PROGRAM PRG_VALVES
VAR
    //Rough lines VRC external interlocks
    bROUGH1_VRC_01_ILK : BOOL;
    bROUGH2_VRC_01_ILK : BOOL;
    bROUGH2_VRC_02_ILK : BOOL;
    bROUGH1_VRC_01_Override : BOOL;
    bROUGH2_VRC_01_Override : BOOL;
    bROUGH2_VRC_02_Override : BOOL;
    bCAT1_VRC_01_ILK : BOOL;
    bDP1_VRC_01_ILK : BOOL;
    bDP1_VRC_02_ILK : BOOL;

    bCAT1_DisableDiffIlk : BOOL;

    //dummy FF output to use in VGC_2S function
    dummy_FFFO : FB_HardwareFFOutput;
    dummy_fbArbiter1 : FB_Arbiter(1);
END_VAR

(**Gas Injection Valves**)
DREAM_DP1_VRC_01(i_stUSG := DREAM_NC_GPI_01.PG,
                 i_stDSG := DREAM_DP1_GPI_01.PG,
                 i_xDis_DPIlk := FALSE,
                 i_xEPS_OK := TRUE,
                 i_xPMPS_OK := TRUE,
                 i_xReset := FALSE,
                 i_xExt_OK := TRUE,
                 i_xOverrideMode := bSystemOverrideMode,
                 io_fbFFHWO := dummy_FFFO,
                 fbArbiter := dummy_fbArbiter1,
                 i_sDevName := 'DREAM-DP1-VRC-01');

//DP1_VRC_02 Interlock evaluation NOTE: Normally OPEN Valve!!
bDP1_VRC_02_ILK := DREAM_DP1_VRC_01.iq_stValve.i_xOpnLS; //Interlock changed for this valve to only gets interlocked by DREAM_DP1_VRC_01 valve

DREAM_DP1_VRC_02(i_xExtILK_OK := bDP1_VRC_02_ILK, i_xOverrideMode := bSystemOverrideMode); //Normally open valve

(**Catcher valve**)
//Evaluate if Diff Interlock is disabled
bCAT1_DisableDiffIlk := NOT GVL_VAC_GAUGES.stDREAM_MC_GAUGE.xPRESS_OK OR NOT DREAM_CAT1_GHC_01.IG.xPRESS_OK;

//CAT1_VRC_01 Interlock evaluation
IF bCAT1_DisableDiffIlk THEN
    bCAT1_VRC_01_ILK := bMCPumpsRunning AND bCATPumpsRunning AND
                        ((GVL_VAC_GAUGES.stDREAM_MC_GAUGE.xPRESS_OK AND GVL_VAC_GAUGES.stDREAM_MC_GAUGE.rPRESS < 5e-4) OR (DREAM_MC_GPI_01.PG.xPRESS_OK AND DREAM_MC_GPI_01.PG.rPRESS < 5e-4)) AND
                        ((DREAM_CAT1_GHC_01.IG.xPRESS_OK AND DREAM_CAT1_GHC_01.IG.rPRESS < 5e-4) OR (DREAM_ROUGH2_GPI_03.PG.xPRESS_OK AND DREAM_ROUGH2_GPI_03.PG.rPRESS < 1e-3));
ELSE
    bCAT1_VRC_01_ILK := bCATPumpsRunning;
END_IF

//DREAM_CAT1_VRC_01(i_xExtILK_OK := bCAT1_VRC_01_ILK, i_xOverrideMode := bSystemOverrideMode);
DREAM_CAT1_VRC_01(i_stUSG := GVL_VAC_GAUGES.stDREAM_MC_GAUGE,
                  i_stDSG := DREAM_CAT1_GHC_01.IG,
                  i_xDis_DPIlk := bCAT1_DisableDiffIlk,
                  i_xEPS_OK := TRUE,
                  i_xPMPS_OK := TRUE,
                  i_xReset := FALSE,
                  i_xExt_OK := bCAT1_VRC_01_ILK,
                  i_xOverrideMode := bSystemOverrideMode,
                  io_fbFFHWO := dummy_FFFO,
                  fbArbiter := dummy_fbArbiter1,
                  i_sDevName := 'DREAM-CAT1-VRC-01');

(**Roughing Valves**)
//Interlock evaluation
bROUGH1_VRC_01_ILK := //DREAM_ROUGH1_GPI_01.PG.rPRESS < 5E-3 AND DREAM_ROUGH1_GPI_01.PG.xPRESS_OK AND
                      DREAM_ROUGH1_VFV_01.iq_stVFN.rReqPosition = 0.0 AND
                      DREAM_ROUGH1_VFV_02.iq_stVFN.rReqPosition = 0.0 AND
                      DREAM_ROUGH1_VRC_10.iq_stValve.i_xClsLS; //Interlocked with manifold roughing valve as well

bROUGH2_VRC_01_ILK := //DREAM_ROUGH2_GPI_01.PG.rPRESS < 5E-3 AND DREAM_ROUGH2_GPI_01.PG.xPRESS_OK AND
                      DREAM_ROUGH2_VFV_01.iq_stVFN.rReqPosition = 0.0 AND
                      DREAM_ROUGH2_VFV_02.iq_stVFN.rReqPosition = 0.0;

bROUGH2_VRC_02_ILK := //DREAM_ROUGH2_GPI_01.PG.rPRESS < 5E-3 AND DREAM_ROUGH2_GPI_01.PG.xPRESS_OK AND
                      DREAM_ROUGH2_VFV_01.iq_stVFN.rReqPosition = 0.0 AND
                      DREAM_ROUGH2_VFV_03.iq_stVFN.rReqPosition = 0.0;

bROUGH1_VRC_01_Override := bSystemOverrideMode AND
                           DREAM_ROUGH1_VFV_01.iq_stVFN.rReqPosition = 0.0 AND
                           DREAM_ROUGH1_VFV_02.iq_stVFN.rReqPosition = 0.0;

bROUGH2_VRC_01_Override := bSystemOverrideMode AND
                           DREAM_ROUGH2_VFV_01.iq_stVFN.rReqPosition = 0.0 AND
                           DREAM_ROUGH2_VFV_02.iq_stVFN.rReqPosition = 0.0;

bROUGH2_VRC_02_Override := bSystemOverrideMode AND
                           DREAM_ROUGH2_VFV_01.iq_stVFN.rReqPosition = 0.0 AND
                           DREAM_ROUGH2_VFV_03.iq_stVFN.rReqPosition = 0.0;

DREAM_ROUGH1_VRC_01(i_stUSG := DREAM_ROUGH1_GPI_01.PG,
                    i_stDSG := DREAM_ROUGH1_GPI_02.PG,
                    i_xDis_DPIlk := FALSE,
                    i_xEPS_OK := TRUE,
                    i_xPMPS_OK := TRUE,
                    i_xReset := FALSE,
                    i_xExt_OK := bROUGH1_VRC_01_ILK,
                    i_xOverrideMode := bROUGH1_VRC_01_Override,
                    io_fbFFHWO := dummy_FFFO,
                    fbArbiter := dummy_fbArbiter1,
                    i_sDevName := 'DREAM-ROUGH1-VRC-01');

DREAM_ROUGH2_VRC_01(i_stUSG := DREAM_ROUGH2_GPI_01.PG,
                    i_stDSG := DREAM_ROUGH2_GPI_02.PG,
                    i_xDis_DPIlk := FALSE,
                    i_xEPS_OK := TRUE,
                    i_xPMPS_OK := TRUE,
                    i_xReset := FALSE,
                    i_xExt_OK := bROUGH2_VRC_01_ILK,
                    i_xOverrideMode := bROUGH2_VRC_01_Override,
                    io_fbFFHWO := dummy_FFFO,
                    fbArbiter := dummy_fbArbiter1,
                    i_sDevName := 'DREAM-ROUGH2-VRC-01');

DREAM_ROUGH2_VRC_02(i_stUSG := DREAM_ROUGH2_GPI_01.PG,
                    i_stDSG := DREAM_ROUGH2_GPI_03.PG,
                    i_xDis_DPIlk := FALSE,
                    i_xEPS_OK := TRUE,
                    i_xPMPS_OK := TRUE,
                    i_xReset := FALSE,
                    i_xExt_OK := bROUGH2_VRC_02_ILK,
                    i_xOverrideMode := bROUGH2_VRC_02_Override,
                    io_fbFFHWO := dummy_FFFO,
                    fbArbiter := dummy_fbArbiter1,
                    i_sDevName := 'DREAM-ROUGH2-VRC-02');

//Test valve
DREAM_ROUGH1_VRC_20(i_xExtILK_OK := True, i_xOverrideMode := bSystemOverrideMode);

//Manifold roughing valve
DREAM_ROUGH1_VRC_10(i_xExtILK_OK := DREAM_ROUGH1_VRC_01.iq_stValve.i_xClsLS, i_xOverrideMode := bSystemOverrideMode);

//Flow control valves
DREAM_ROUGH1_VFV_01(i_xExtIlkOK := DREAM_ROUGH1_VRC_01.iq_stValve.i_xClsLS);

DREAM_ROUGH1_VFV_02(i_xExtIlkOK := DREAM_ROUGH1_VRC_01.iq_stValve.i_xClsLS AND DREAM_DP1_VRC_01.iq_stValve.i_xClsLS AND
                                   NOT DREAM_NC_PTM_01.iq_stPTM.i_xAtSpd AND
                                   NOT DREAM_NC_PTM_02.iq_stPTM.i_xAtSpd);

DREAM_ROUGH2_VFV_01(i_xExtIlkOK := DREAM_ROUGH2_VRC_01.iq_stValve.i_xClsLS AND DREAM_ROUGH2_VRC_02.iq_stValve.i_xClsLS);

DREAM_ROUGH2_VFV_02(i_xExtIlkOK := DREAM_ROUGH2_VRC_01.iq_stValve.i_xClsLS AND
                                   NOT DREAM_DP1_PTM_01.iq_stPTM.i_xAtSpd AND
                                   NOT DREAM_DP2_PTM_01.iq_stPTM.i_xAtSpd AND
                                   NOT DREAM_DP3_PTM_01.iq_stPTM.i_xAtSpd AND
                                   NOT DREAM_MC_PTM_01.iq_stPTM.i_xAtSpd AND
                                   NOT DREAM_MC_PTM_02.iq_stPTM.i_xAtSpd AND
                                   NOT DREAM_ROUGH2_PTM_01.iq_stPTM.i_xAtSpd AND
                                   NOT DREAM_ROUGH2_PTM_02.iq_stPTM.i_xAtSpd AND
                                   NOT DREAM_CAT1_PTM_01.iq_stPTM.i_xAtSpd);

DREAM_ROUGH2_VFV_03(i_xExtIlkOK := DREAM_ROUGH2_VRC_02.iq_stValve.i_xClsLS AND DREAM_CAT1_VRC_01.iq_stValve.i_xClsLS AND
                                   NOT DREAM_CAT2_PTM_01.iq_stPtm.i_xAtSpd);

END_PROGRAM

(* stored: Version 1.1.0.1, ProductVersion 3.1.4024.12
   POU PRG_VALVES: Id {03dcac03-cfad-4254-831b-855af8503ea4}, SpecialFunc None *)
